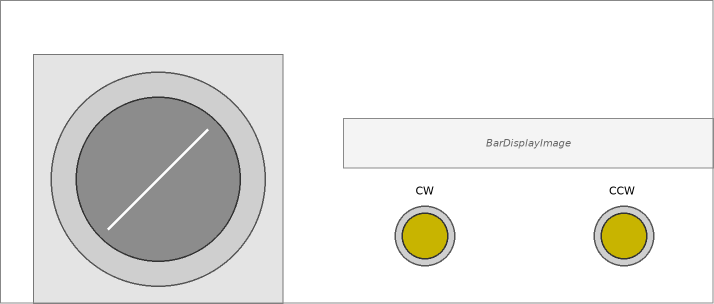
VISUALIZATION Visualization_reference  // 714x304
    Potentiometer360 (33,54 250x250), variable: Input.iHMISlide, style: Potentiometer-Potentiometer360-Gray, scale format: %.1f, scale -660..660
        p2431819421: Outside
    BarDisplayImage (343,118 371x50), value: MR_J_Motor.iInVoltage, style: BarDisplayImage-Gray, scale format: %.1f, scale 0..660
    Lamp1 (390,201 70x70), variable: MR_J_Motor.bCW, style: Lamp-Lamp1-Yellow
    Lamp1 (589,201 70x70), variable: MR_J_Motor.bCCW, style: Lamp-Lamp1-Yellow
    Label (350,176 150x30), "CW"
    Label (547,176 150x30), "CCW"
END_VISUALIZATION

(* stored: Version 1.1.0.1, ProductVersion 3.1.4026.6
   Visu Visualization_reference: Id {2643f7ea-71ce-42f8-ba58-c71b2da8999c} *)
